SUBAPPLICATION mapping_aux (* Subapplication Type *)
  (* Standard: 61499-2 *)
  (* Version 1.0, 2023-01-29, Franz *)
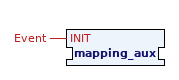
  EVENT_INPUT
    INIT;
  END_EVENT
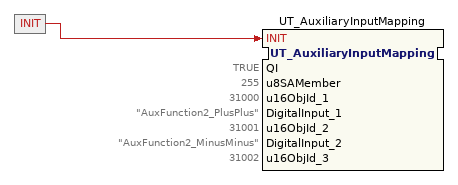
  FBS
    UT_AuxiliaryInputMapping : UT_AuxiliaryInputMapping(QI := TRUE, u8SAMember := 255, u16ObjId_1 := 31000, DigitalInput_1 := "AuxFunction2_PlusPlus", u16ObjId_2 := 31001, DigitalInput_2 := "AuxFunction2_MinusMinus", u16ObjId_3 := 31002);
  END_FBS
  EVENT_CONNECTIONS
    INIT TO UT_AuxiliaryInputMapping.INIT;
  END_CONNECTIONS
END_SUBAPPLICATION
